(* CoDeSys 2.3.9.62 project: Ampelsteuerung.pro *)
(* Libraries: Standard.lib, IecSfc.lib 2.6.14 10:37:46, SYSLIBCALLBACK.LIB *)

(* Global variable list: Globale_Variablen *)
VAR_GLOBAL
	E1: BOOL;
	E2: BOOL;
END_VAR

(* POU PLC_PRG, FBD *)
PROGRAM PLC_PRG
VAR
END_VAR
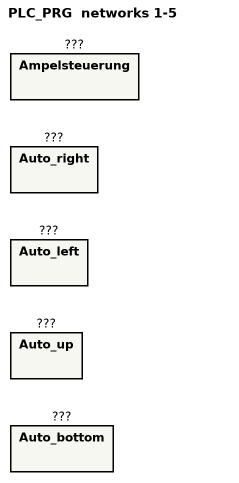
_FBD_ (* Function Block Diagram *)
NETWORK 1
	???:Ampelsteuerung()
NETWORK 2
	???:Auto_right()
NETWORK 3
	???:Auto_left()
NETWORK 4
	???:Auto_up()
NETWORK 5
	???:Auto_bottom()
_END_FBD_
END_PROGRAM

(* POU Ampelsteuerung, SFC *)
PROGRAM Ampelsteuerung
VAR
	Start: BOOL;
	Stop:BOOL;

	H_ROT:BOOL;
	H_GELB:BOOL;
	H_GRUEN:BOOL;

	N_ROT:BOOL;
	N_GELB:BOOL;
	N_GRUEN:BOOL;


	START_TRIGGER: R_TRIG;
	Start_Phasen_Timer: TON;
	Start_HGelb: TON;
	Start_NGelb: TON;
	Start_STimer1: BOOL;
	Start_STimer2: BOOL;

	Phase_GELB: TON;
	Phase_ROT: TON;
	Phase_HROT_HGELB: TON;
	Phase_HGRUEN: TON;
	Phase_HGRUEN_1: TON;
	Phase_HGELB: TON;
	Phase_HROT: TON;
	Phase_NROT_NGELB: TON;
	Phase_NGRUEN: TON;
	Phase_NGELB: TON;

END_VAR
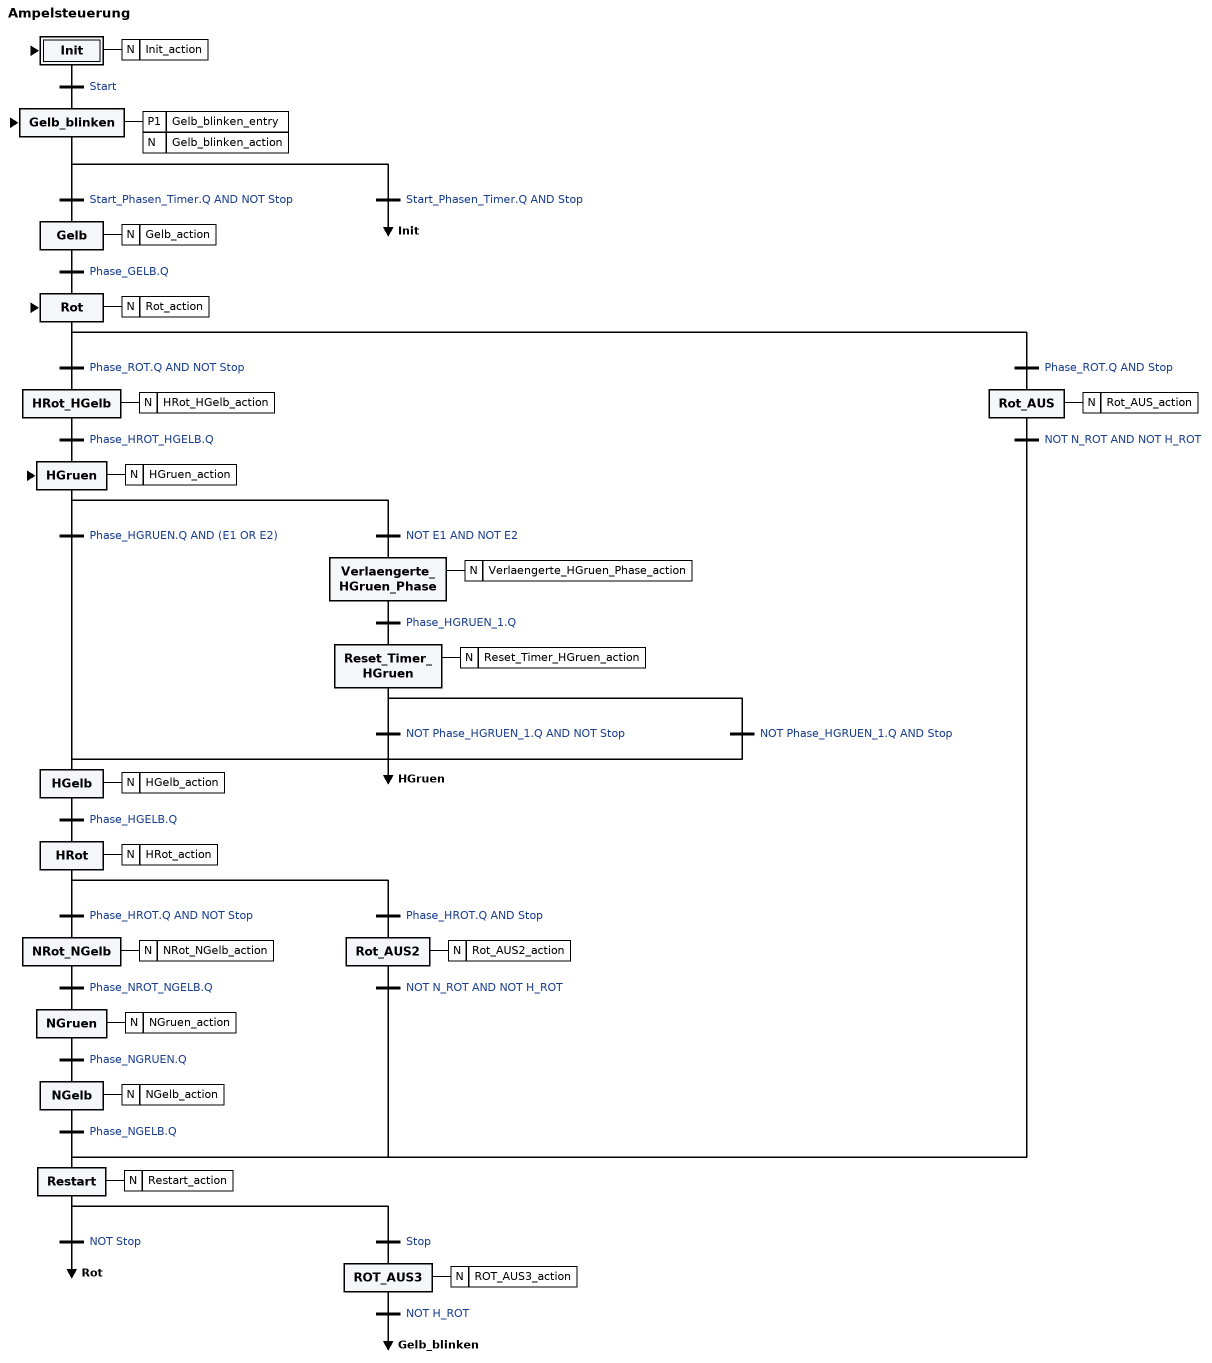
INITIAL_STEP Init:
	Init_action(N);
END_STEP
TRANSITION FROM Init TO Gelb_blinken := Start;
END_TRANSITION
STEP Gelb_blinken:
	Gelb_blinken_entry(P1);
	Gelb_blinken_action(N);
END_STEP
TRANSITION FROM Gelb_blinken TO Gelb := Start_Phasen_Timer.Q AND NOT Stop;
END_TRANSITION
TRANSITION FROM Gelb_blinken TO Init := Start_Phasen_Timer.Q AND Stop;
END_TRANSITION
STEP Gelb:
	Gelb_action(N);
END_STEP
TRANSITION FROM Gelb TO Rot := Phase_GELB.Q;
END_TRANSITION
STEP Rot:
	Rot_action(N);
END_STEP
TRANSITION FROM Rot TO HRot_HGelb := Phase_ROT.Q AND NOT Stop;
END_TRANSITION
TRANSITION FROM Rot TO Rot_AUS := Phase_ROT.Q AND Stop;
END_TRANSITION
STEP Rot_AUS:
	Rot_AUS_action(N);
END_STEP
TRANSITION FROM Rot_AUS TO Restart := NOT N_ROT AND NOT H_ROT;
END_TRANSITION
STEP HRot_HGelb:
	HRot_HGelb_action(N);
END_STEP
TRANSITION FROM HRot_HGelb TO HGruen := Phase_HROT_HGELB.Q;
END_TRANSITION
STEP HGruen:
	HGruen_action(N);
END_STEP
TRANSITION FROM HGruen TO HGelb := Phase_HGRUEN.Q AND (E1 OR E2);
END_TRANSITION
TRANSITION FROM HGruen TO Verlaengerte_HGruen_Phase := NOT E1 AND NOT E2;
END_TRANSITION
STEP Verlaengerte_HGruen_Phase:
	Verlaengerte_HGruen_Phase_action(N);
END_STEP
TRANSITION FROM Verlaengerte_HGruen_Phase TO Reset_Timer_HGruen := Phase_HGRUEN_1.Q;
END_TRANSITION
STEP Reset_Timer_HGruen:
	Reset_Timer_HGruen_action(N);
END_STEP
TRANSITION FROM Reset_Timer_HGruen TO HGruen := NOT Phase_HGRUEN_1.Q AND NOT Stop;
END_TRANSITION
TRANSITION FROM Reset_Timer_HGruen TO HGelb := NOT Phase_HGRUEN_1.Q AND Stop;
END_TRANSITION
STEP HGelb:
	HGelb_action(N);
END_STEP
TRANSITION FROM HGelb TO HRot := Phase_HGELB.Q;
END_TRANSITION
STEP HRot:
	HRot_action(N);
END_STEP
TRANSITION FROM HRot TO NRot_NGelb := Phase_HROT.Q AND NOT Stop;
END_TRANSITION
TRANSITION FROM HRot TO Rot_AUS2 := Phase_HROT.Q AND Stop;
END_TRANSITION
STEP Rot_AUS2:
	Rot_AUS2_action(N);
END_STEP
TRANSITION FROM Rot_AUS2 TO Restart := NOT N_ROT AND NOT H_ROT;
END_TRANSITION
STEP NRot_NGelb:
	NRot_NGelb_action(N);
END_STEP
TRANSITION FROM NRot_NGelb TO NGruen := Phase_NROT_NGELB.Q;
END_TRANSITION
STEP NGruen:
	NGruen_action(N);
END_STEP
TRANSITION FROM NGruen TO NGelb := Phase_NGRUEN.Q;
END_TRANSITION
STEP NGelb:
	NGelb_action(N);
END_STEP
TRANSITION FROM NGelb TO Restart := Phase_NGELB.Q;
END_TRANSITION
STEP Restart:
	Restart_action(N);
END_STEP
TRANSITION FROM Restart TO Rot := NOT Stop;
END_TRANSITION
TRANSITION FROM Restart TO ROT_AUS3 := Stop;
END_TRANSITION
STEP ROT_AUS3:
	ROT_AUS3_action(N);
END_STEP
TRANSITION FROM ROT_AUS3 TO Gelb_blinken := NOT H_ROT;
END_TRANSITION

ACTION Init_action:
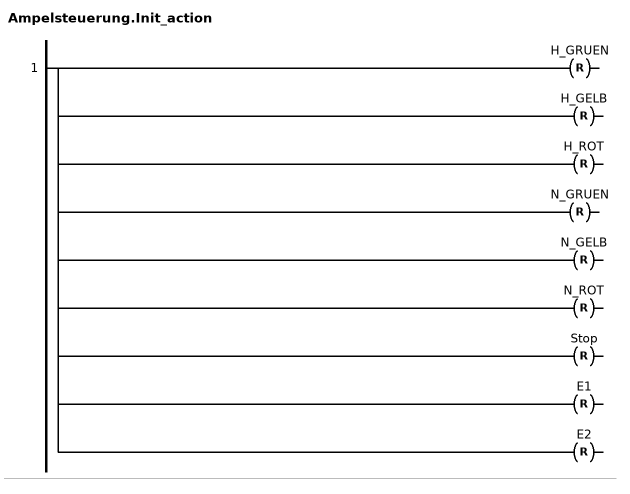
_LD_ (* Ladder Diagram *)
NETWORK 1
	* --- (R H_GRUEN) (R H_GELB) (R H_ROT) (R N_GRUEN) (R N_GELB) (R N_ROT) (R Stop) (R E1) (R E2)
_END_LD_
(* the same logic as Structured Text *)
(* Network 1 *)
H_GRUEN := FALSE;
H_GELB := FALSE;
H_ROT := FALSE;
N_GRUEN := FALSE;
N_GELB := FALSE;
N_ROT := FALSE;
Stop := FALSE;
E1 := FALSE;
E2 := FALSE;
END_ACTION

ACTION Gelb_blinken_entry:
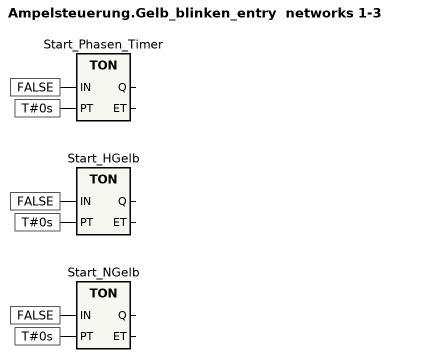
_FBD_ (* Function Block Diagram *)
NETWORK 1
	Start_Phasen_Timer:TON(IN: FALSE, PT: T#0s)
NETWORK 2
	Start_HGelb:TON(IN: FALSE, PT: T#0s)
NETWORK 3
	Start_NGelb:TON(IN: FALSE, PT: T#0s)
_END_FBD_
(* the same logic as Structured Text *)
(* Network 1 *)
Start_Phasen_Timer(IN := FALSE, PT := T#0s);
(* Network 2 *)
Start_HGelb(IN := FALSE, PT := T#0s);
(* Network 3 *)
Start_NGelb(IN := FALSE, PT := T#0s);
END_ACTION

ACTION Gelb_blinken_action:
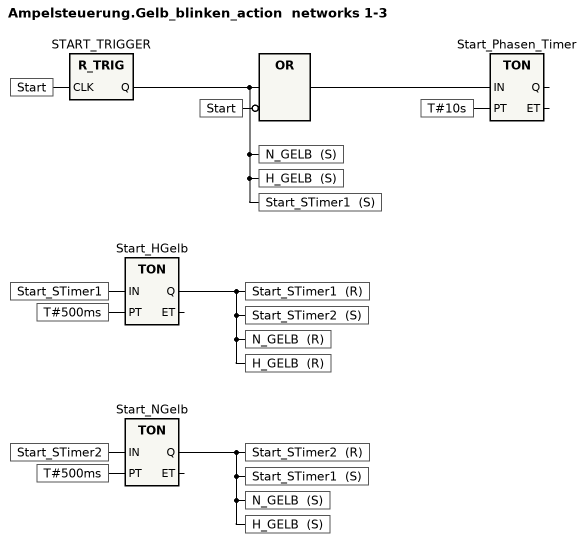
_FBD_ (* Function Block Diagram *)
NETWORK 1
	Start_Phasen_Timer:TON(IN: OR(<<<START_TRIGGER:R_TRIG(CLK: Start) => S N_GELB> => S H_GELB> => S Start_STimer1>, NOT Start), PT: T#10s)
NETWORK 2
	<<<Start_HGelb:TON(IN: Start_STimer1, PT: T#500ms) => R Start_STimer1> => S Start_STimer2> => R N_GELB> => R H_GELB
NETWORK 3
	<<<Start_NGelb:TON(IN: Start_STimer2, PT: T#500ms) => R Start_STimer2> => S Start_STimer1> => S N_GELB> => S H_GELB
_END_FBD_
(* the same logic as Structured Text *)
(* Network 1 *)
START_TRIGGER(CLK := Start);
IF START_TRIGGER.Q THEN N_GELB := TRUE; END_IF;
IF START_TRIGGER.Q THEN H_GELB := TRUE; END_IF;
IF START_TRIGGER.Q THEN Start_STimer1 := TRUE; END_IF;
Start_Phasen_Timer(IN := START_TRIGGER.Q OR NOT Start, PT := T#10s);
(* Network 2 *)
Start_HGelb(IN := Start_STimer1, PT := T#500ms);
IF Start_HGelb.Q THEN Start_STimer1 := FALSE; END_IF;
IF Start_HGelb.Q THEN Start_STimer2 := TRUE; END_IF;
IF Start_HGelb.Q THEN N_GELB := FALSE; END_IF;
IF Start_HGelb.Q THEN H_GELB := FALSE; END_IF;
(* Network 3 *)
Start_NGelb(IN := Start_STimer2, PT := T#500ms);
IF Start_NGelb.Q THEN Start_STimer2 := FALSE; END_IF;
IF Start_NGelb.Q THEN Start_STimer1 := TRUE; END_IF;
IF Start_NGelb.Q THEN N_GELB := TRUE; END_IF;
IF Start_NGelb.Q THEN H_GELB := TRUE; END_IF;
END_ACTION

ACTION Gelb_action:
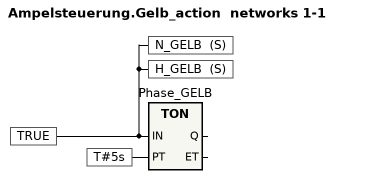
_FBD_ (* Function Block Diagram *)
NETWORK 1
	Phase_GELB:TON(IN: <<TRUE => S N_GELB> => S H_GELB>, PT: T#5s)
_END_FBD_
(* the same logic as Structured Text *)
(* Network 1 *)
N_GELB := TRUE;
H_GELB := TRUE;
Phase_GELB(IN := TRUE, PT := T#5s);
END_ACTION

ACTION Rot_action:
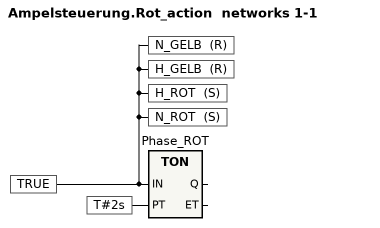
_FBD_ (* Function Block Diagram *)
NETWORK 1
	Phase_ROT:TON(IN: <<<<TRUE => R N_GELB> => R H_GELB> => S H_ROT> => S N_ROT>, PT: T#2s)
_END_FBD_
(* the same logic as Structured Text *)
(* Network 1 *)
N_GELB := FALSE;
H_GELB := FALSE;
H_ROT := TRUE;
N_ROT := TRUE;
Phase_ROT(IN := TRUE, PT := T#2s);
END_ACTION

ACTION Rot_AUS_action:
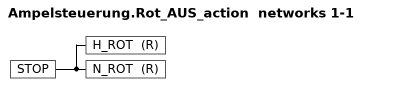
_FBD_ (* Function Block Diagram *)
NETWORK 1
	<STOP => R H_ROT> => R N_ROT
_END_FBD_
(* the same logic as Structured Text *)
(* Network 1 *)
IF STOP THEN H_ROT := FALSE; END_IF;
IF STOP THEN N_ROT := FALSE; END_IF;
END_ACTION

ACTION HRot_HGelb_action:
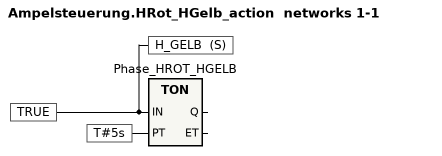
_FBD_ (* Function Block Diagram *)
NETWORK 1
	Phase_HROT_HGELB:TON(IN: <TRUE => S H_GELB>, PT: T#5s)
_END_FBD_
(* the same logic as Structured Text *)
(* Network 1 *)
H_GELB := TRUE;
Phase_HROT_HGELB(IN := TRUE, PT := T#5s);
END_ACTION

ACTION HGruen_action:
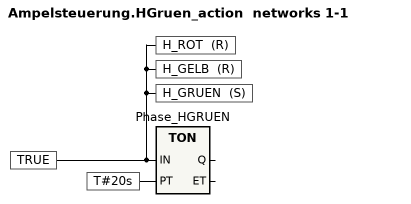
_FBD_ (* Function Block Diagram *)
NETWORK 1
	Phase_HGRUEN:TON(IN: <<<TRUE => R H_ROT> => R H_GELB> => S H_GRUEN>, PT: T#20s)
_END_FBD_
(* the same logic as Structured Text *)
(* Network 1 *)
H_ROT := FALSE;
H_GELB := FALSE;
H_GRUEN := TRUE;
Phase_HGRUEN(IN := TRUE, PT := T#20s);
END_ACTION

ACTION Verlaengerte_HGruen_Phase_action:
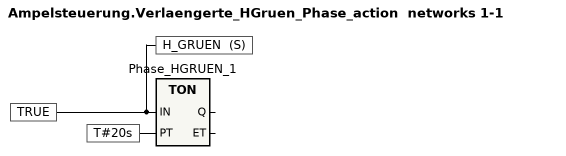
_FBD_ (* Function Block Diagram *)
NETWORK 1
	Phase_HGRUEN_1:TON(IN: <TRUE => S H_GRUEN>, PT: T#20s)
_END_FBD_
(* the same logic as Structured Text *)
(* Network 1 *)
H_GRUEN := TRUE;
Phase_HGRUEN_1(IN := TRUE, PT := T#20s);
END_ACTION

ACTION Reset_Timer_HGruen_action:
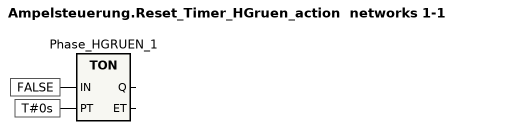
_FBD_ (* Function Block Diagram *)
NETWORK 1
	Phase_HGRUEN_1:TON(IN: FALSE, PT: T#0s)
_END_FBD_
(* the same logic as Structured Text *)
(* Network 1 *)
Phase_HGRUEN_1(IN := FALSE, PT := T#0s);
END_ACTION

ACTION HGelb_action:
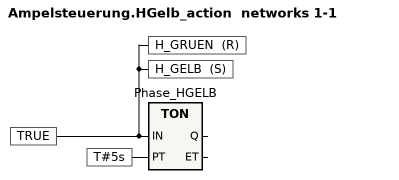
_FBD_ (* Function Block Diagram *)
NETWORK 1
	Phase_HGELB:TON(IN: <<TRUE => R H_GRUEN> => S H_GELB>, PT: T#5s)
_END_FBD_
(* the same logic as Structured Text *)
(* Network 1 *)
H_GRUEN := FALSE;
H_GELB := TRUE;
Phase_HGELB(IN := TRUE, PT := T#5s);
END_ACTION

ACTION HRot_action:
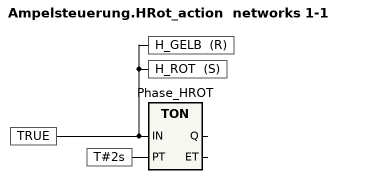
_FBD_ (* Function Block Diagram *)
NETWORK 1
	Phase_HROT:TON(IN: <<TRUE => R H_GELB> => S H_ROT>, PT: T#2s)
_END_FBD_
(* the same logic as Structured Text *)
(* Network 1 *)
H_GELB := FALSE;
H_ROT := TRUE;
Phase_HROT(IN := TRUE, PT := T#2s);
END_ACTION

ACTION Rot_AUS2_action:
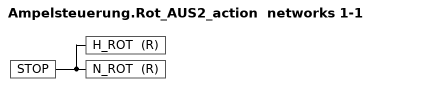
_FBD_ (* Function Block Diagram *)
NETWORK 1
	<STOP => R H_ROT> => R N_ROT
_END_FBD_
(* the same logic as Structured Text *)
(* Network 1 *)
IF STOP THEN H_ROT := FALSE; END_IF;
IF STOP THEN N_ROT := FALSE; END_IF;
END_ACTION

ACTION NRot_NGelb_action:
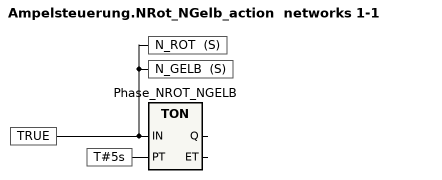
_FBD_ (* Function Block Diagram *)
NETWORK 1
	Phase_NROT_NGELB:TON(IN: <<TRUE => S N_ROT> => S N_GELB>, PT: T#5s)
_END_FBD_
(* the same logic as Structured Text *)
(* Network 1 *)
N_ROT := TRUE;
N_GELB := TRUE;
Phase_NROT_NGELB(IN := TRUE, PT := T#5s);
END_ACTION

ACTION NGruen_action:
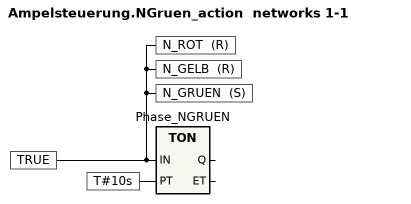
_FBD_ (* Function Block Diagram *)
NETWORK 1
	Phase_NGRUEN:TON(IN: <<<TRUE => R N_ROT> => R N_GELB> => S N_GRUEN>, PT: T#10s)
_END_FBD_
(* the same logic as Structured Text *)
(* Network 1 *)
N_ROT := FALSE;
N_GELB := FALSE;
N_GRUEN := TRUE;
Phase_NGRUEN(IN := TRUE, PT := T#10s);
END_ACTION

ACTION NGelb_action:
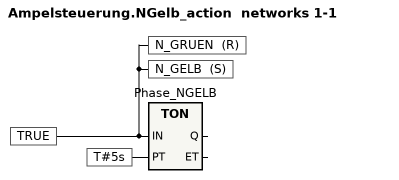
_FBD_ (* Function Block Diagram *)
NETWORK 1
	Phase_NGELB:TON(IN: <<TRUE => R N_GRUEN> => S N_GELB>, PT: T#5s)
_END_FBD_
(* the same logic as Structured Text *)
(* Network 1 *)
N_GRUEN := FALSE;
N_GELB := TRUE;
Phase_NGELB(IN := TRUE, PT := T#5s);
END_ACTION

ACTION Restart_action:
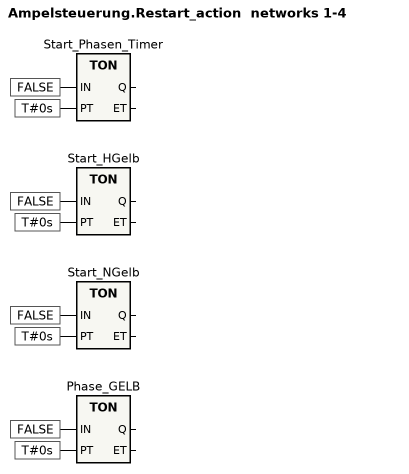
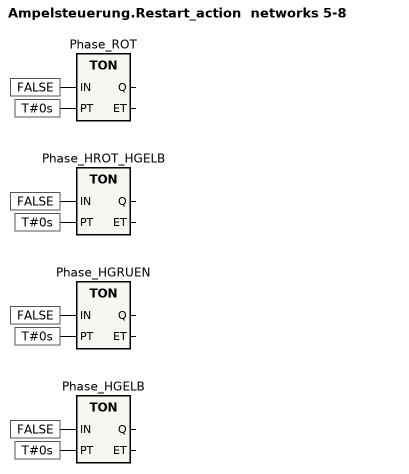
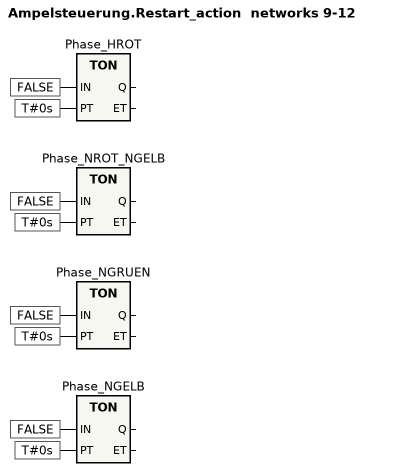
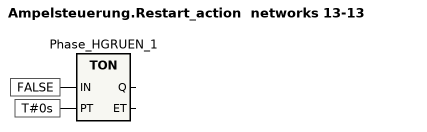
_FBD_ (* Function Block Diagram *)
NETWORK 1
	Start_Phasen_Timer:TON(IN: FALSE, PT: T#0s)
NETWORK 2
	Start_HGelb:TON(IN: FALSE, PT: T#0s)
NETWORK 3
	Start_NGelb:TON(IN: FALSE, PT: T#0s)
NETWORK 4
	Phase_GELB:TON(IN: FALSE, PT: T#0s)
NETWORK 5
	Phase_ROT:TON(IN: FALSE, PT: T#0s)
NETWORK 6
	Phase_HROT_HGELB:TON(IN: FALSE, PT: T#0s)
NETWORK 7
	Phase_HGRUEN:TON(IN: FALSE, PT: T#0s)
NETWORK 8
	Phase_HGELB:TON(IN: FALSE, PT: T#0s)
NETWORK 9
	Phase_HROT:TON(IN: FALSE, PT: T#0s)
NETWORK 10
	Phase_NROT_NGELB:TON(IN: FALSE, PT: T#0s)
NETWORK 11
	Phase_NGRUEN:TON(IN: FALSE, PT: T#0s)
NETWORK 12
	Phase_NGELB:TON(IN: FALSE, PT: T#0s)
NETWORK 13
	Phase_HGRUEN_1:TON(IN: FALSE, PT: T#0s)
_END_FBD_
(* the same logic as Structured Text *)
(* Network 1 *)
Start_Phasen_Timer(IN := FALSE, PT := T#0s);
(* Network 2 *)
Start_HGelb(IN := FALSE, PT := T#0s);
(* Network 3 *)
Start_NGelb(IN := FALSE, PT := T#0s);
(* Network 4 *)
Phase_GELB(IN := FALSE, PT := T#0s);
(* Network 5 *)
Phase_ROT(IN := FALSE, PT := T#0s);
(* Network 6 *)
Phase_HROT_HGELB(IN := FALSE, PT := T#0s);
(* Network 7 *)
Phase_HGRUEN(IN := FALSE, PT := T#0s);
(* Network 8 *)
Phase_HGELB(IN := FALSE, PT := T#0s);
(* Network 9 *)
Phase_HROT(IN := FALSE, PT := T#0s);
(* Network 10 *)
Phase_NROT_NGELB(IN := FALSE, PT := T#0s);
(* Network 11 *)
Phase_NGRUEN(IN := FALSE, PT := T#0s);
(* Network 12 *)
Phase_NGELB(IN := FALSE, PT := T#0s);
(* Network 13 *)
Phase_HGRUEN_1(IN := FALSE, PT := T#0s);
END_ACTION

ACTION ROT_AUS3_action:
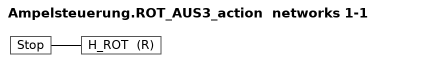
_FBD_ (* Function Block Diagram *)
NETWORK 1
	Stop => R H_ROT
_END_FBD_
(* the same logic as Structured Text *)
(* Network 1 *)
IF Stop THEN H_ROT := FALSE; END_IF;
END_ACTION
END_PROGRAM

(* POU Auto_right, ST *)
PROGRAM Auto_right
VAR
	car_east: INT:=0;
	a: INT;
END_VAR
IF car_east > -240 AND car_east < -230 AND Ampelsteuerung.H_ROT THEN
;
ELSE
car_east := car_east - 5;
END_IF

IF car_east < -650 THEN
car_east := 0;
END_IF
END_PROGRAM

(* POU Auto_left, ST *)
PROGRAM Auto_left
VAR
	car_west: INT:= 0;
END_VAR
IF car_west < 240 AND car_west > 230 AND Ampelsteuerung.H_ROT THEN
;
ELSE
car_west:= car_west + 5;
END_IF

IF car_west > 640 THEN
car_west := 0;
END_IF
END_PROGRAM

(* POU Auto_up, ST *)
PROGRAM Auto_up
VAR
	car_nord: INT:= 0;
END_VAR
IF car_nord <200 AND car_nord > 190 AND NOT Ampelsteuerung.N_GRUEN THEN
E1 := TRUE;
ELSE
E1 :=FALSE;
car_nord := car_nord + 5;
END_IF

IF car_nord > 650 THEN
car_nord := 0;
END_IF
END_PROGRAM

(* POU Auto_bottom, ST *)
PROGRAM Auto_bottom
VAR
	car_south: INT :=0;
END_VAR
IF car_south > -235 AND car_south < -225 AND NOT Ampelsteuerung.N_GRUEN THEN
E2:= TRUE;
ELSE
E2:=FALSE;
car_south:= car_south - 5;
END_IF

IF car_south < -650 THEN
car_south := 0;
END_IF
END_PROGRAM

(* Visualisation Kreuzung
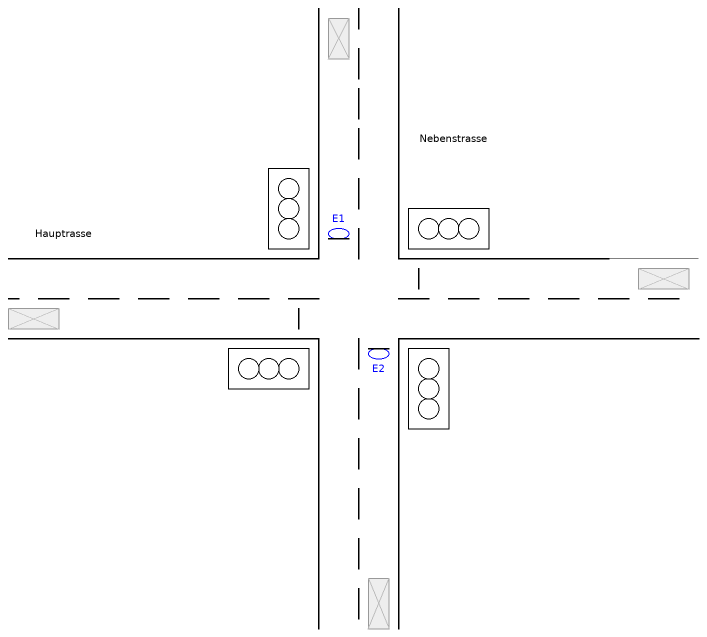
ellipse at (380,220)-(401,241): alarm colour if Ampelsteuerung.N_GRUEN
ellipse at (380,240)-(401,261): alarm colour if Ampelsteuerung.N_GELB
ellipse at (380,260)-(401,281): alarm colour if Ampelsteuerung.N_ROT
ellipse at (520,260)-(541,281): alarm colour if Ampelsteuerung.H_ROT
ellipse at (540,260)-(561,281): alarm colour if Ampelsteuerung.H_GELB
ellipse at (560,260)-(581,281): alarm colour if Ampelsteuerung.H_GRUEN
ellipse at (380,400)-(401,421): alarm colour if Ampelsteuerung.H_ROT
ellipse at (360,400)-(381,421): alarm colour if Ampelsteuerung.H_GELB
ellipse at (520,440)-(541,461): alarm colour if Ampelsteuerung.N_GRUEN
ellipse at (520,420)-(541,441): alarm colour if Ampelsteuerung.N_GELB
ellipse at (520,400)-(541,421): alarm colour if Ampelsteuerung.N_ROT
ellipse at (340,400)-(361,421): alarm colour if Ampelsteuerung.H_GRUEN
rectangle at (500,170)-(611,191): text "Nebenstrasse"
rectangle at (110,260)-(221,291): text "Hauptrasse"
rounded rectangle at (430,250)-(451,271): text "E1"
rectangle at (470,400)-(491,421): text "E2"
bitmap at (740,310)-(791,331): auto_rechts.bmp
bitmap at (430,60)-(451,101): polizei.bmp
bitmap at (110,350)-(161,371): auto_links.bmp
bitmap at (470,620)-(491,671): krankenwagen.bmp
57 more shapes without text or variables
*)

(* Visualisation Zustaende
